{attribute 'qualified_only'}
VAR_GLOBAL
	//theme:NtkR5fYqIUM
	//test:dutDWord;
	memtype:INT; // I,Q,M,etc
	memsize:INT; //number of bytes, 8, 16, 32
	memswap:INT; //swap endianness 
	memHexDisplay:INT; //swap endianness 



	btnLower: BOOL;
	btnLowerFaster: BOOL;
	btnRaise: BOOL;
	btnRaiseFaster: BOOL;

	row01:dutDWord;
	row02:dutDWord;
	row03:dutDWord;
	row04:dutDWord;
	row05:dutDWord;
	row06:dutDWord;
	row07:dutDWord;
	row08:dutDWord;
	row09:dutDWord;
	row10:dutDWord;
	row11:dutDWord;
	row12:dutDWord;
	row13:dutDWord;
	row14:dutDWord;
	row15:dutDWord;
	row16:dutDWord;
	
	ByteRow: ARRAY[0..15] OF dutDWord;

	//deposit data from mempointer
	ViewingArray: ARRAY[0..32] OF DWORD;
	memoffset:UDINT;
	
	blockNum:SINT;

END_VAR

(* stored: Version 1.1.0.1, ProductVersion 3.1.4024.12
   GVL ioView: Id {8e54282d-4c10-4d90-abf2-2b5c8eaa87f3} *)
